# EPICS substitutions: apps/caenHvApp/Db/subs/HVDC2_DC_4527.substitutions
#
#This file was autogenerated by mkHVEpics.C on: Wed Nov  2 16:01:55 2016
#Substitutions for crate: HVDC2,  detector: DC
#
file "db/caenhv.db" {
        pattern { Cr,    CrName,         CrType, Sl,     Ch,    Sys,     Det,    Element,                CScode, pwonoff, v0set,  i0set,   trip,    rampup,  rampdn, svmax,   enable, dark}
		{"13",	"HVDC2",	"1527",	"00",	"00",	"HV",	"DC",	"SEC5_R1_SL1_S01-08",	"#C13", "S2816", "S512", "S1280", "S2560", "S1024", "S768", "S3328", "S256", "1"}
		{"13",	"HVDC2",	"1527",	"00",	"01",	"HV",	"DC",	"SEC5_R1_SL1_S09-16",	"#C13", "S2817", "S513", "S1281", "S2561", "S1025", "S769", "S3329", "S257", "1"}
		{"13",	"HVDC2",	"1527",	"00",	"02",	"HV",	"DC",	"SEC5_R1_SL1_S17-24",	"#C13", "S2818", "S514", "S1282", "S2562", "S1026", "S770", "S3330", "S258", "1"}
		{"13",	"HVDC2",	"1527",	"00",	"03",	"HV",	"DC",	"SEC5_R1_SL1_S25-32",	"#C13", "S2819", "S515", "S1283", "S2563", "S1027", "S771", "S3331", "S259", "1"}
		{"13",	"HVDC2",	"1527",	"00",	"04",	"HV",	"DC",	"SEC5_R1_SL1_S33-48",	"#C13", "S2820", "S516", "S1284", "S2564", "S1028", "S772", "S3332", "S260", "1"}
		{"13",	"HVDC2",	"1527",	"00",	"05",	"HV",	"DC",	"SEC5_R1_SL1_S49-64",	"#C13", "S2821", "S517", "S1285", "S2565", "S1029", "S773", "S3333", "S261", "1"}
		{"13",	"HVDC2",	"1527",	"00",	"06",	"HV",	"DC",	"SEC5_R1_SL1_S65-80",	"#C13", "S2822", "S518", "S1286", "S2566", "S1030", "S774", "S3334", "S262", "1"}
		{"13",	"HVDC2",	"1527",	"00",	"07",	"HV",	"DC",	"SEC5_R1_SL1_S81-112",	"#C13", "S2823", "S519", "S1287", "S2567", "S1031", "S775", "S3335", "S263", "1"}
		{"13",	"HVDC2",	"1527",	"00",	"08",	"HV",	"DC",	"SEC5_R1_SL2_S01-08",	"#C13", "S2824", "S520", "S1288", "S2568", "S1032", "S776", "S3336", "S264", "1"}
		{"13",	"HVDC2",	"1527",	"00",	"09",	"HV",	"DC",	"SEC5_R1_SL2_S09-16",	"#C13", "S2825", "S521", "S1289", "S2569", "S1033", "S777", "S3337", "S265", "1"}
		{"13",	"HVDC2",	"1527",	"00",	"10",	"HV",	"DC",	"SEC5_R1_SL2_S17-24",	"#C13", "S2826", "S522", "S1290", "S2570", "S1034", "S778", "S3338", "S266", "1"}
		{"13",	"HVDC2",	"1527",	"00",	"11",	"HV",	"DC",	"SEC5_R1_SL2_S25-32",	"#C13", "S2827", "S523", "S1291", "S2571", "S1035", "S779", "S3339", "S267", "1"}
		{"13",	"HVDC2",	"1527",	"00",	"12",	"HV",	"DC",	"SEC5_R1_SL2_S33-48",	"#C13", "S2828", "S524", "S1292", "S2572", "S1036", "S780", "S3340", "S268", "1"}
		{"13",	"HVDC2",	"1527",	"00",	"13",	"HV",	"DC",	"SEC5_R1_SL2_S49-64",	"#C13", "S2829", "S525", "S1293", "S2573", "S1037", "S781", "S3341", "S269", "1"}
		{"13",	"HVDC2",	"1527",	"00",	"14",	"HV",	"DC",	"SEC5_R1_SL2_S65-80",	"#C13", "S2830", "S526", "S1294", "S2574", "S1038", "S782", "S3342", "S270", "1"}
		{"13",	"HVDC2",	"1527",	"00",	"15",	"HV",	"DC",	"SEC5_R1_SL2_S81-112",	"#C13", "S2831", "S527", "S1295", "S2575", "S1039", "S783", "S3343", "S271", "1"}
		{"13",	"HVDC2",	"1527",	"00",	"16",	"HV",	"DC",	"SEC4_R1_SL1_S01-08",	"#C13", "S2832", "S528", "S1296", "S2576", "S1040", "S784", "S3344", "S272", "1"}
		{"13",	"HVDC2",	"1527",	"00",	"17",	"HV",	"DC",	"SEC4_R1_SL1_S09-16",	"#C13", "S2833", "S529", "S1297", "S2577", "S1041", "S785", "S3345", "S273", "1"}
		{"13",	"HVDC2",	"1527",	"00",	"18",	"HV",	"DC",	"SEC4_R1_SL1_S17-24",	"#C13", "S2834", "S530", "S1298", "S2578", "S1042", "S786", "S3346", "S274", "1"}
		{"13",	"HVDC2",	"1527",	"00",	"19",	"HV",	"DC",	"SEC4_R1_SL1_S25-32",	"#C13", "S2835", "S531", "S1299", "S2579", "S1043", "S787", "S3347", "S275", "1"}
		{"13",	"HVDC2",	"1527",	"00",	"20",	"HV",	"DC",	"SEC4_R1_SL1_S33-48",	"#C13", "S2836", "S532", "S1300", "S2580", "S1044", "S788", "S3348", "S276", "1"}
		{"13",	"HVDC2",	"1527",	"00",	"21",	"HV",	"DC",	"SEC4_R1_SL1_S49-64",	"#C13", "S2837", "S533", "S1301", "S2581", "S1045", "S789", "S3349", "S277", "1"}
		{"13",	"HVDC2",	"1527",	"00",	"22",	"HV",	"DC",	"SEC4_R1_SL1_S65-80",	"#C13", "S2838", "S534", "S1302", "S2582", "S1046", "S790", "S3350", "S278", "1"}
		{"13",	"HVDC2",	"1527",	"00",	"23",	"HV",	"DC",	"SEC4_R1_SL1_S81-112",	"#C13", "S2839", "S535", "S1303", "S2583", "S1047", "S791", "S3351", "S279", "1"}
		{"13",	"HVDC2",	"1527",	"01",	"00",	"HV",	"DC",	"SEC4_R1_SL2_S01-08",	"#C269", "S2816", "S512", "S1280", "S2560", "S1024", "S768", "S3328", "S256", "1"}
		{"13",	"HVDC2",	"1527",	"01",	"01",	"HV",	"DC",	"SEC4_R1_SL2_S09-16",	"#C269", "S2817", "S513", "S1281", "S2561", "S1025", "S769", "S3329", "S257", "1"}
		{"13",	"HVDC2",	"1527",	"01",	"02",	"HV",	"DC",	"SEC4_R1_SL2_S17-24",	"#C269", "S2818", "S514", "S1282", "S2562", "S1026", "S770", "S3330", "S258", "1"}
		{"13",	"HVDC2",	"1527",	"01",	"03",	"HV",	"DC",	"SEC4_R1_SL2_S25-32",	"#C269", "S2819", "S515", "S1283", "S2563", "S1027", "S771", "S3331", "S259", "1"}
		{"13",	"HVDC2",	"1527",	"01",	"04",	"HV",	"DC",	"SEC4_R1_SL2_S33-48",	"#C269", "S2820", "S516", "S1284", "S2564", "S1028", "S772", "S3332", "S260", "1"}
		{"13",	"HVDC2",	"1527",	"01",	"05",	"HV",	"DC",	"SEC4_R1_SL2_S49-64",	"#C269", "S2821", "S517", "S1285", "S2565", "S1029", "S773", "S3333", "S261", "1"}
		{"13",	"HVDC2",	"1527",	"01",	"06",	"HV",	"DC",	"SEC4_R1_SL2_S65-80",	"#C269", "S2822", "S518", "S1286", "S2566", "S1030", "S774", "S3334", "S262", "1"}
		{"13",	"HVDC2",	"1527",	"01",	"07",	"HV",	"DC",	"SEC4_R1_SL2_S81-112",	"#C269", "S2823", "S519", "S1287", "S2567", "S1031", "S775", "S3335", "S263", "1"}
		{"13",	"HVDC2",	"1527",	"01",	"08",	"HV",	"DC",	"SEC3_R1_SL1_S01-08",	"#C269", "S2824", "S520", "S1288", "S2568", "S1032", "S776", "S3336", "S264", "1"}
		{"13",	"HVDC2",	"1527",	"01",	"09",	"HV",	"DC",	"SEC3_R1_SL1_S09-16",	"#C269", "S2825", "S521", "S1289", "S2569", "S1033", "S777", "S3337", "S265", "1"}
		{"13",	"HVDC2",	"1527",	"01",	"10",	"HV",	"DC",	"SEC3_R1_SL1_S17-24",	"#C269", "S2826", "S522", "S1290", "S2570", "S1034", "S778", "S3338", "S266", "1"}
		{"13",	"HVDC2",	"1527",	"01",	"11",	"HV",	"DC",	"SEC3_R1_SL1_S25-32",	"#C269", "S2827", "S523", "S1291", "S2571", "S1035", "S779", "S3339", "S267", "1"}
		{"13",	"HVDC2",	"1527",	"01",	"12",	"HV",	"DC",	"SEC3_R1_SL1_S33-48",	"#C269", "S2828", "S524", "S1292", "S2572", "S1036", "S780", "S3340", "S268", "1"}
		{"13",	"HVDC2",	"1527",	"01",	"13",	"HV",	"DC",	"SEC3_R1_SL1_S49-64",	"#C269", "S2829", "S525", "S1293", "S2573", "S1037", "S781", "S3341", "S269", "1"}
		{"13",	"HVDC2",	"1527",	"01",	"14",	"HV",	"DC",	"SEC3_R1_SL1_S65-80",	"#C269", "S2830", "S526", "S1294", "S2574", "S1038", "S782", "S3342", "S270", "1"}
		{"13",	"HVDC2",	"1527",	"01",	"15",	"HV",	"DC",	"SEC3_R1_SL1_S81-112",	"#C269", "S2831", "S527", "S1295", "S2575", "S1039", "S783", "S3343", "S271", "1"}
		{"13",	"HVDC2",	"1527",	"01",	"16",	"HV",	"DC",	"SEC3_R1_SL2_S01-08",	"#C269", "S2832", "S528", "S1296", "S2576", "S1040", "S784", "S3344", "S272", "1"}
		{"13",	"HVDC2",	"1527",	"01",	"17",	"HV",	"DC",	"SEC3_R1_SL2_S09-16",	"#C269", "S2833", "S529", "S1297", "S2577", "S1041", "S785", "S3345", "S273", "1"}
		{"13",	"HVDC2",	"1527",	"01",	"18",	"HV",	"DC",	"SEC3_R1_SL2_S17-24",	"#C269", "S2834", "S530", "S1298", "S2578", "S1042", "S786", "S3346", "S274", "1"}
		{"13",	"HVDC2",	"1527",	"01",	"19",	"HV",	"DC",	"SEC3_R1_SL2_S25-32",	"#C269", "S2835", "S531", "S1299", "S2579", "S1043", "S787", "S3347", "S275", "1"}
		{"13",	"HVDC2",	"1527",	"01",	"20",	"HV",	"DC",	"SEC3_R1_SL2_S33-48",	"#C269", "S2836", "S532", "S1300", "S2580", "S1044", "S788", "S3348", "S276", "1"}
		{"13",	"HVDC2",	"1527",	"01",	"21",	"HV",	"DC",	"SEC3_R1_SL2_S49-64",	"#C269", "S2837", "S533", "S1301", "S2581", "S1045", "S789", "S3349", "S277", "1"}
		{"13",	"HVDC2",	"1527",	"01",	"22",	"HV",	"DC",	"SEC3_R1_SL2_S65-80",	"#C269", "S2838", "S534", "S1302", "S2582", "S1046", "S790", "S3350", "S278", "1"}
		{"13",	"HVDC2",	"1527",	"01",	"23",	"HV",	"DC",	"SEC3_R1_SL2_S81-112",	"#C269", "S2839", "S535", "S1303", "S2583", "S1047", "S791", "S3351", "S279", "1"}
		{"13",	"HVDC2",	"1527",	"02",	"00",	"HV",	"DC",	"SEC5_R1_SL1_F01-08",	"#C525", "S2816", "S512", "S1280", "S2560", "S1024", "S768", "S3328", "S256", "1"}
		{"13",	"HVDC2",	"1527",	"02",	"01",	"HV",	"DC",	"SEC5_R1_SL1_F09-16",	"#C525", "S2817", "S513", "S1281", "S2561", "S1025", "S769", "S3329", "S257", "1"}
		{"13",	"HVDC2",	"1527",	"02",	"02",	"HV",	"DC",	"SEC5_R1_SL1_F17-24",	"#C525", "S2818", "S514", "S1282", "S2562", "S1026", "S770", "S3330", "S258", "1"}
		{"13",	"HVDC2",	"1527",	"02",	"03",	"HV",	"DC",	"SEC5_R1_SL1_F25-32",	"#C525", "S2819", "S515", "S1283", "S2563", "S1027", "S771", "S3331", "S259", "1"}
		{"13",	"HVDC2",	"1527",	"02",	"04",	"HV",	"DC",	"SEC5_R1_SL1_F33-48",	"#C525", "S2820", "S516", "S1284", "S2564", "S1028", "S772", "S3332", "S260", "1"}
		{"13",	"HVDC2",	"1527",	"02",	"05",	"HV",	"DC",	"SEC5_R1_SL1_F49-64",	"#C525", "S2821", "S517", "S1285", "S2565", "S1029", "S773", "S3333", "S261", "1"}
		{"13",	"HVDC2",	"1527",	"02",	"06",	"HV",	"DC",	"SEC5_R1_SL1_F65-80",	"#C525", "S2822", "S518", "S1286", "S2566", "S1030", "S774", "S3334", "S262", "1"}
		{"13",	"HVDC2",	"1527",	"02",	"07",	"HV",	"DC",	"SEC5_R1_SL1_F81-112",	"#C525", "S2823", "S519", "S1287", "S2567", "S1031", "S775", "S3335", "S263", "1"}
		{"13",	"HVDC2",	"1527",	"02",	"08",	"HV",	"DC",	"SEC5_R1_SL2_F01-08",	"#C525", "S2824", "S520", "S1288", "S2568", "S1032", "S776", "S3336", "S264", "1"}
		{"13",	"HVDC2",	"1527",	"02",	"09",	"HV",	"DC",	"SEC5_R1_SL2_F09-16",	"#C525", "S2825", "S521", "S1289", "S2569", "S1033", "S777", "S3337", "S265", "1"}
		{"13",	"HVDC2",	"1527",	"02",	"10",	"HV",	"DC",	"SEC5_R1_SL2_F17-24",	"#C525", "S2826", "S522", "S1290", "S2570", "S1034", "S778", "S3338", "S266", "1"}
		{"13",	"HVDC2",	"1527",	"02",	"11",	"HV",	"DC",	"SEC5_R1_SL2_F25-32",	"#C525", "S2827", "S523", "S1291", "S2571", "S1035", "S779", "S3339", "S267", "1"}
		{"13",	"HVDC2",	"1527",	"02",	"12",	"HV",	"DC",	"SEC5_R1_SL2_F33-48",	"#C525", "S2828", "S524", "S1292", "S2572", "S1036", "S780", "S3340", "S268", "1"}
		{"13",	"HVDC2",	"1527",	"02",	"13",	"HV",	"DC",	"SEC5_R1_SL2_F49-64",	"#C525", "S2829", "S525", "S1293", "S2573", "S1037", "S781", "S3341", "S269", "1"}
		{"13",	"HVDC2",	"1527",	"02",	"14",	"HV",	"DC",	"SEC5_R1_SL2_F65-80",	"#C525", "S2830", "S526", "S1294", "S2574", "S1038", "S782", "S3342", "S270", "1"}
		{"13",	"HVDC2",	"1527",	"02",	"15",	"HV",	"DC",	"SEC5_R1_SL2_F81-112",	"#C525", "S2831", "S527", "S1295", "S2575", "S1039", "S783", "S3343", "S271", "1"}
		{"13",	"HVDC2",	"1527",	"02",	"16",	"HV",	"DC",	"SEC4_R1_SL1_F01-08",	"#C525", "S2832", "S528", "S1296", "S2576", "S1040", "S784", "S3344", "S272", "1"}
		{"13",	"HVDC2",	"1527",	"02",	"17",	"HV",	"DC",	"SEC4_R1_SL1_F09-16",	"#C525", "S2833", "S529", "S1297", "S2577", "S1041", "S785", "S3345", "S273", "1"}
		{"13",	"HVDC2",	"1527",	"02",	"18",	"HV",	"DC",	"SEC4_R1_SL1_F17-24",	"#C525", "S2834", "S530", "S1298", "S2578", "S1042", "S786", "S3346", "S274", "1"}
		{"13",	"HVDC2",	"1527",	"02",	"19",	"HV",	"DC",	"SEC4_R1_SL1_F25-32",	"#C525", "S2835", "S531", "S1299", "S2579", "S1043", "S787", "S3347", "S275", "1"}
		{"13",	"HVDC2",	"1527",	"02",	"20",	"HV",	"DC",	"SEC4_R1_SL1_F33-48",	"#C525", "S2836", "S532", "S1300", "S2580", "S1044", "S788", "S3348", "S276", "1"}
		{"13",	"HVDC2",	"1527",	"02",	"21",	"HV",	"DC",	"SEC4_R1_SL1_F49-64",	"#C525", "S2837", "S533", "S1301", "S2581", "S1045", "S789", "S3349", "S277", "1"}
		{"13",	"HVDC2",	"1527",	"02",	"22",	"HV",	"DC",	"SEC4_R1_SL1_F65-80",	"#C525", "S2838", "S534", "S1302", "S2582", "S1046", "S790", "S3350", "S278", "1"}
		{"13",	"HVDC2",	"1527",	"02",	"23",	"HV",	"DC",	"SEC4_R1_SL1_F81-112",	"#C525", "S2839", "S535", "S1303", "S2583", "S1047", "S791", "S3351", "S279", "1"}
		{"13",	"HVDC2",	"1527",	"03",	"00",	"HV",	"DC",	"SEC4_R1_SL2_F01-08",	"#C781", "S2816", "S512", "S1280", "S2560", "S1024", "S768", "S3328", "S256", "1"}
		{"13",	"HVDC2",	"1527",	"03",	"01",	"HV",	"DC",	"SEC4_R1_SL2_F09-16",	"#C781", "S2817", "S513", "S1281", "S2561", "S1025", "S769", "S3329", "S257", "1"}
		{"13",	"HVDC2",	"1527",	"03",	"02",	"HV",	"DC",	"SEC4_R1_SL2_F17-24",	"#C781", "S2818", "S514", "S1282", "S2562", "S1026", "S770", "S3330", "S258", "1"}
		{"13",	"HVDC2",	"1527",	"03",	"03",	"HV",	"DC",	"SEC4_R1_SL2_F25-32",	"#C781", "S2819", "S515", "S1283", "S2563", "S1027", "S771", "S3331", "S259", "1"}
		{"13",	"HVDC2",	"1527",	"03",	"04",	"HV",	"DC",	"SEC4_R1_SL2_F33-48",	"#C781", "S2820", "S516", "S1284", "S2564", "S1028", "S772", "S3332", "S260", "1"}
		{"13",	"HVDC2",	"1527",	"03",	"05",	"HV",	"DC",	"SEC4_R1_SL2_F49-64",	"#C781", "S2821", "S517", "S1285", "S2565", "S1029", "S773", "S3333", "S261", "1"}
		{"13",	"HVDC2",	"1527",	"03",	"06",	"HV",	"DC",	"SEC4_R1_SL2_F65-80",	"#C781", "S2822", "S518", "S1286", "S2566", "S1030", "S774", "S3334", "S262", "1"}
		{"13",	"HVDC2",	"1527",	"03",	"07",	"HV",	"DC",	"SEC4_R1_SL2_F81-112",	"#C781", "S2823", "S519", "S1287", "S2567", "S1031", "S775", "S3335", "S263", "1"}
		{"13",	"HVDC2",	"1527",	"03",	"08",	"HV",	"DC",	"SEC3_R1_SL1_F01-08",	"#C781", "S2824", "S520", "S1288", "S2568", "S1032", "S776", "S3336", "S264", "1"}
		{"13",	"HVDC2",	"1527",	"03",	"09",	"HV",	"DC",	"SEC3_R1_SL1_F09-16",	"#C781", "S2825", "S521", "S1289", "S2569", "S1033", "S777", "S3337", "S265", "1"}
		{"13",	"HVDC2",	"1527",	"03",	"10",	"HV",	"DC",	"SEC3_R1_SL1_F17-24",	"#C781", "S2826", "S522", "S1290", "S2570", "S1034", "S778", "S3338", "S266", "1"}
		{"13",	"HVDC2",	"1527",	"03",	"11",	"HV",	"DC",	"SEC3_R1_SL1_F25-32",	"#C781", "S2827", "S523", "S1291", "S2571", "S1035", "S779", "S3339", "S267", "1"}
		{"13",	"HVDC2",	"1527",	"03",	"12",	"HV",	"DC",	"SEC3_R1_SL1_F33-48",	"#C781", "S2828", "S524", "S1292", "S2572", "S1036", "S780", "S3340", "S268", "1"}
		{"13",	"HVDC2",	"1527",	"03",	"13",	"HV",	"DC",	"SEC3_R1_SL1_F49-64",	"#C781", "S2829", "S525", "S1293", "S2573", "S1037", "S781", "S3341", "S269", "1"}
		{"13",	"HVDC2",	"1527",	"03",	"14",	"HV",	"DC",	"SEC3_R1_SL1_F65-80",	"#C781", "S2830", "S526", "S1294", "S2574", "S1038", "S782", "S3342", "S270", "1"}
		{"13",	"HVDC2",	"1527",	"03",	"15",	"HV",	"DC",	"SEC3_R1_SL1_F81-112",	"#C781", "S2831", "S527", "S1295", "S2575", "S1039", "S783", "S3343", "S271", "1"}
		{"13",	"HVDC2",	"1527",	"03",	"16",	"HV",	"DC",	"SEC3_R1_SL2_F01-08",	"#C781", "S2832", "S528", "S1296", "S2576", "S1040", "S784", "S3344", "S272", "1"}
		{"13",	"HVDC2",	"1527",	"03",	"17",	"HV",	"DC",	"SEC3_R1_SL2_F09-16",	"#C781", "S2833", "S529", "S1297", "S2577", "S1041", "S785", "S3345", "S273", "1"}
		{"13",	"HVDC2",	"1527",	"03",	"18",	"HV",	"DC",	"SEC3_R1_SL2_F17-24",	"#C781", "S2834", "S530", "S1298", "S2578", "S1042", "S786", "S3346", "S274", "1"}
		{"13",	"HVDC2",	"1527",	"03",	"19",	"HV",	"DC",	"SEC3_R1_SL2_F25-32",	"#C781", "S2835", "S531", "S1299", "S2579", "S1043", "S787", "S3347", "S275", "1"}
		{"13",	"HVDC2",	"1527",	"03",	"20",	"HV",	"DC",	"SEC3_R1_SL2_F33-48",	"#C781", "S2836", "S532", "S1300", "S2580", "S1044", "S788", "S3348", "S276", "1"}
		{"13",	"HVDC2",	"1527",	"03",	"21",	"HV",	"DC",	"SEC3_R1_SL2_F49-64",	"#C781", "S2837", "S533", "S1301", "S2581", "S1045", "S789", "S3349", "S277", "1"}
		{"13",	"HVDC2",	"1527",	"03",	"22",	"HV",	"DC",	"SEC3_R1_SL2_F65-80",	"#C781", "S2838", "S534", "S1302", "S2582", "S1046", "S790", "S3350", "S278", "1"}
		{"13",	"HVDC2",	"1527",	"03",	"23",	"HV",	"DC",	"SEC3_R1_SL2_F81-112",	"#C781", "S2839", "S535", "S1303", "S2583", "S1047", "S791", "S3351", "S279", "1"}
		{"13",	"HVDC2",	"1527",	"04",	"00",	"HV",	"DC",	"SEC5_R1_SL1_G01-32",	"#C1037", "S2816", "S512", "S1280", "S2560", "S1024", "S768", "S3328", "S256", "1"}
		{"13",	"HVDC2",	"1527",	"04",	"01",	"HV",	"DC",	"SEC5_R1_SL1_G33-112",	"#C1037", "S2817", "S513", "S1281", "S2561", "S1025", "S769", "S3329", "S257", "1"}
		{"13",	"HVDC2",	"1527",	"04",	"02",	"HV",	"DC",	"SEC5_R1_SL2_G01-32",	"#C1037", "S2818", "S514", "S1282", "S2562", "S1026", "S770", "S3330", "S258", "1"}
		{"13",	"HVDC2",	"1527",	"04",	"03",	"HV",	"DC",	"SEC5_R1_SL2_G33-112",	"#C1037", "S2819", "S515", "S1283", "S2563", "S1027", "S771", "S3331", "S259", "1"}
		{"13",	"HVDC2",	"1527",	"04",	"04",	"HV",	"DC",	"SEC4_R1_SL1_G01-32",	"#C1037", "S2820", "S516", "S1284", "S2564", "S1028", "S772", "S3332", "S260", "1"}
		{"13",	"HVDC2",	"1527",	"04",	"05",	"HV",	"DC",	"SEC4_R1_SL1_G33-112",	"#C1037", "S2821", "S517", "S1285", "S2565", "S1029", "S773", "S3333", "S261", "1"}
		{"13",	"HVDC2",	"1527",	"04",	"06",	"HV",	"DC",	"SEC4_R1_SL2_G01-32",	"#C1037", "S2822", "S518", "S1286", "S2566", "S1030", "S774", "S3334", "S262", "1"}
		{"13",	"HVDC2",	"1527",	"04",	"07",	"HV",	"DC",	"SEC4_R1_SL2_G33-112",	"#C1037", "S2823", "S519", "S1287", "S2567", "S1031", "S775", "S3335", "S263", "1"}
		{"13",	"HVDC2",	"1527",	"04",	"08",	"HV",	"DC",	"SEC3_R1_SL1_G01-32",	"#C1037", "S2824", "S520", "S1288", "S2568", "S1032", "S776", "S3336", "S264", "1"}
		{"13",	"HVDC2",	"1527",	"04",	"09",	"HV",	"DC",	"SEC3_R1_SL1_G33-112",	"#C1037", "S2825", "S521", "S1289", "S2569", "S1033", "S777", "S3337", "S265", "1"}
		{"13",	"HVDC2",	"1527",	"04",	"10",	"HV",	"DC",	"SEC3_R1_SL2_G01-32",	"#C1037", "S2826", "S522", "S1290", "S2570", "S1034", "S778", "S3338", "S266", "1"}
		{"13",	"HVDC2",	"1527",	"04",	"11",	"HV",	"DC",	"SEC3_R1_SL2_G33-112",	"#C1037", "S2827", "S523", "S1291", "S2571", "S1035", "S779", "S3339", "S267", "1"}
}
